// TIA Portal project "PLCUnit" (V15)

(* hardware
DEVICE "S71500/ET200MP station_1"  S7-1500 station
   slot 0: "Rail_0"  Rack  6ES7 590-1***0-0AA0
   slot 1: "PLC_1"  CPU 1511-1 PN  6ES7 511-1AK02-0AB0  V2.5
      slot 3: "CPU display_1"  6ES7591-1AA00-0AA0
   slot 2: "AI 8xU/I/RTD/TC ST_1"  AI 8xU/I/RTD/TC ST  6ES7 531-7KF00-0AB0  V2.1
   slot 3: "AI 8xU/I/RTD/TC ST_2"  AI 8xU/I/RTD/TC ST  6ES7 531-7KF00-0AB0  V2.1
   slot 4: "AI 8xU/I/RTD/TC ST_3"  AI 8xU/I/RTD/TC ST  6ES7 531-7KF00-0AB0  V2.1
   slot 5: "AI 8xU/I/RTD/TC ST_4"  AI 8xU/I/RTD/TC ST  6ES7 531-7KF00-0AB0  V2.1
   slot 6: "DI 16x24VDC BA_1"  DI 16x24VDC BA  6ES7 521-1BH10-0AA0  V1.0
   slot 7: "DQ 16x24VDC/0.5A BA_1"  DQ 16x24VDC/0.5A BA  6ES7 522-1BH10-0AA0  V1.0
*)

// ===== PLC "PLC_1"  CPU 1511-1 PN =====

VAR_GLOBAL   // PLC tag table "Default tag table"
   "DO_1" AT %Q514.0 : Bool;
   "DI_1" AT %I512.0 : Bool;
   "Tag_1" AT %Q0.0 : Bool;
END_VAR

DATA_BLOCK "Default_SupervisionDB"   // DB1
{ S7_Optimized_Access := 'TRUE' }
VERSION : 0.1
// stored: InstanceOfName Default_SupervisionFB
"Default_SupervisionFB"
BEGIN
END_DATA_BLOCK

DATA_BLOCK "DI"   // DB2
{ S7_Optimized_Access := 'FALSE' }
VERSION : 0.1
   VAR
      Engine_On_Button : Bool;
      Sensor_Station_1 : Bool;
      Sensor_Station_2 : Bool;
   END_VAR
BEGIN
END_DATA_BLOCK

DATA_BLOCK "Engine_DB"   // DB3
{ S7_Optimized_Access := 'TRUE' }
VERSION : 0.1
// stored: InstanceOfName Engine
"Engine"
BEGIN
END_DATA_BLOCK

DATA_BLOCK "DO"   // DB4
{ S7_Optimized_Access := 'FALSE' }
VERSION : 0.1
   VAR
      Engine : Bool;
      Engine_Station_1 : Bool;
      Engine_Station_2 : Bool;
   END_VAR
BEGIN
END_DATA_BLOCK

DATA_BLOCK "BottleMachine_DB"   // DB5
{ S7_Optimized_Access := 'TRUE' }
VERSION : 0.1
// stored: InstanceOfName BottleMachine
"BottleMachine"
BEGIN
END_DATA_BLOCK

FUNCTION_BLOCK "Engine"   // FB1, LAD
{ S7_Optimized_Access := 'TRUE' }
VERSION : 0.1
BEGIN

REGION Network 1: Turn On Engine
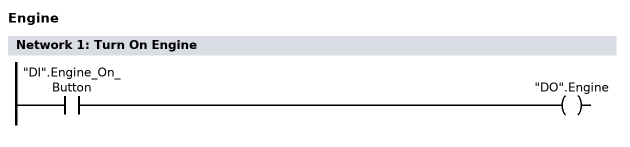
   RUNG wire#powerrail
      Contact( "DI".Engine_On_Button )
      Coil( "DO".Engine )
   END_RUNG
   // the same network as SCL:
   "DO".Engine := "DI".Engine_On_Button;
END_REGION
END_FUNCTION_BLOCK

FUNCTION_BLOCK "Default_SupervisionFB"   // FB2, ProDiag
{ S7_Optimized_Access := 'TRUE' }
   VAR
      PC_Flags : PC_Flags_V2;
      State : SV_FB_State_V2;
   END_VAR
   VAR_TEMP
      t_TempSvStateUDT : SV_State_V2;
      t_TempAlarmInstance : <type 200004f>;
      t_TempAsocValue1 : Variant;
      t_TempAsocValue2 : Variant;
      t_TempAsocValue3 : Variant;
   END_VAR
BEGIN
END_FUNCTION_BLOCK

FUNCTION_BLOCK "BottleMachine"   // FB3, LAD
{ S7_Optimized_Access := 'TRUE' }
VERSION : 0.1
BEGIN

REGION Network 1: Station 1
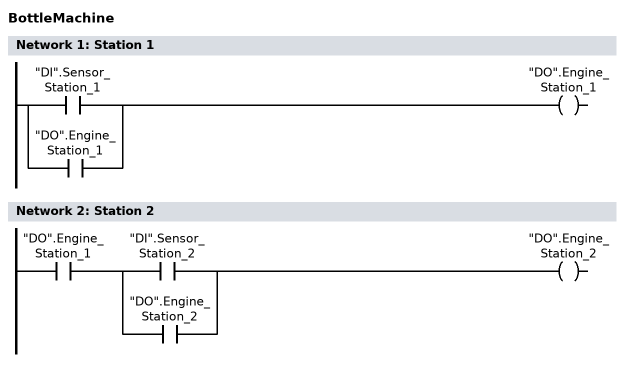
   RUNG wire#powerrail
      Contact( "DI".Sensor_Station_1 )
      wire#w1
      Coil( "DO".Engine_Station_1 )
   END_RUNG
   RUNG wire#powerrail
      Contact( "DO".Engine_Station_1 )
   END_RUNG wire#w1
   // the same network as SCL:
   "DO".Engine_Station_1 := "DI".Sensor_Station_1 OR "DO".Engine_Station_1;
END_REGION

REGION Network 2: Station 2
   RUNG wire#powerrail
      Contact( "DO".Engine_Station_1 )
      wire#w1
      Contact( "DI".Sensor_Station_2 )
      wire#w2
      Coil( "DO".Engine_Station_2 )
   END_RUNG
   RUNG wire#w1
      Contact( "DO".Engine_Station_2 )
   END_RUNG wire#w2
   // the same network as SCL:
   "DO".Engine_Station_2 := "DO".Engine_Station_1 AND ("DI".Sensor_Station_2 OR "DO".Engine_Station_2);
END_REGION
END_FUNCTION_BLOCK

FUNCTION "MHJ-PLC-Lab-Function-S71500" : Void   // FC9000, SCL
{ S7_Optimized_Access := 'FALSE' }
VERSION : 0.1
   VAR_TEMP
      Value : Byte;
      ForCounter : Int;
   END_VAR
   VAR CONSTANT
      Value_01_DW : DWord := 16#1223_5486;
      Value_02_DW : DWord := 16#A6C9_D1F5;
   END_VAR
BEGIN

   #Value := PEEK(area := 16#82,
                  dbNumber := 0,
                  byteOffset := 511);
   #Value := #Value + 1;

   POKE(area := 16#82,
        dbNumber := 0,
        byteOffset := 511,
        value := #Value);

   POKE(area := 16#82,
        dbNumber := 0,
        byteOffset := 1016,
        value := #Value_01_DW);
   POKE(area := 16#82,
        dbNumber := 0,
        byteOffset := 1020,
        value := #Value_02_DW);

   FOR #ForCounter := 0 TO 63 DO
       #Value := PEEK(area := 16#1,
                      dbNumber := 0,
                      byteOffset := #ForCounter);
       POKE(area := 16#81,
            dbNumber := 0,
            byteOffset := #ForCounter,
            value := #Value);
   END_FOR;
   #Value := PEEK(area := 16#1,
                  dbNumber := 0,
                  byteOffset := 512);
   POKE(area := 16#82,
        dbNumber := 0,
        byteOffset := 512,
        value := #Value);
END_FUNCTION

ORGANIZATION_BLOCK "Main"   // OB1, LAD, ProgramCycle
TITLE = "Main Program Sweep (Cycle)"
{ S7_Optimized_Access := 'TRUE' }
VERSION : 0.1
   VAR_INPUT
      Initial_Call : Bool;   // Initial call of this OB
      Remanence : Bool;   // =True, if remanent data are available
   END_VAR
BEGIN

REGION Network 1
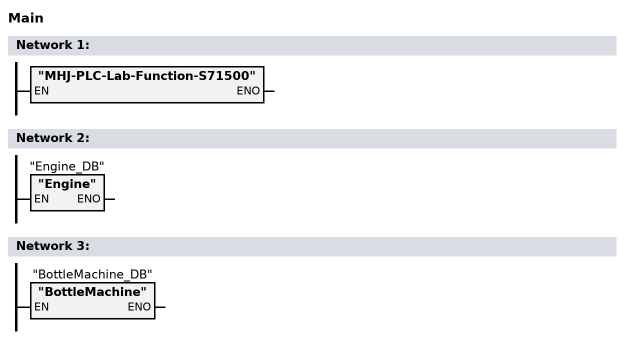
   RUNG wire#powerrail
      "MHJ-PLC-Lab-Function-S71500"()
   END_RUNG
   // the same network as SCL:
   "MHJ-PLC-Lab-Function-S71500"();
END_REGION

REGION Network 2
   RUNG wire#powerrail
      "Engine_DB"()
   END_RUNG
   // the same network as SCL:
   "Engine_DB"();   // "Engine"
END_REGION

REGION Network 3
   RUNG wire#powerrail
      "BottleMachine_DB"()
   END_RUNG
   // the same network as SCL:
   "BottleMachine_DB"();   // "BottleMachine"
END_REGION
END_ORGANIZATION_BLOCK

ORGANIZATION_BLOCK "ProDiagOB"   // OB250, ProDiag_OB, ProgramCycle
TITLE = "Main Program Sweep (Cycle)"
{ S7_Optimized_Access := 'TRUE' }
VERSION : 0.1
   VAR_INPUT
      Initial_Call : Bool;   // Initial call of this OB
      Remanence : Bool;   // =True, if remanent data are available
   END_VAR
BEGIN

REGION Network 1
   CALL "Default_SupervisionFB", "Default_SupervisionDB";
END_REGION
END_ORGANIZATION_BLOCK